FUNCTION AWAIT_ASSERTIONS
VAR_INPUT
    AwaitTime : TIME;
END_VAR
VAR
    IteratorCounter : UINT;
    CurrentTestPointer : POINTER TO FB_Test;
    NumberOfTestsToAnalyse : UINT(1..GVL_Param_TcUnit.MaxNumberOfTestSuites);
END_VAR

GVL_TcUnit.CurrentTestBeingCalled.AwaitingTimer(IN:=TRUE,PT:=AwaitTime);
GVL_TcUnit.CurrentTestBeingCalled.AssertionIsAwaiting := NOT GVL_TcUnit.CurrentTestBeingCalled.AwaitingTimer.Q;

END_FUNCTION

(* stored: Version 1.1.0.1, ProductVersion 3.1.4024.9
   POU AWAIT_ASSERTIONS: Id {1f553859-c334-4de8-8600-188644aee40d}, SpecialFunc None *)
